// TIA Portal V20 export
// export: Created 2025-12-01T14:57:26.6752033Z, ExportSetting None, DisplayName Totally Integrated Automation Portal, DisplayVersion V20 Update 3, DisplayName TIA Portal Openness, DisplayVersion V20 Update 3, DisplayName TIA Portal Version Control Interface, DisplayVersion V20 Update 3, DisplayName STEP 7 Professional, DisplayVersion V20 Update 3, DisplayName STEP 7 Safety, DisplayVersion V20 Update 2, DisplayName WinCC Basic/Comfort/Advanced, DisplayVersion V20 Update 3, DisplayName WinCC Professional, DisplayVersion V20 Update 3, DisplayName WinCC Unified, DisplayVersion V20 Update 3
FUNCTION "FC602_ReservaPeine" : Void   // FC602, LAD
{ S7_Optimized_Access := 'TRUE' }
// stored: AutoNumber false, SetENOAutomatically false
   VAR_INPUT
      ID_Quimarox : UInt;
      ID_ElementoPeticion : UInt;
      TipoDeElemento : UInt;
   END_VAR
   VAR_OUTPUT
      NumeroPeineReservado : UInt;
   END_VAR
   VAR_TEMP
      PeineParaReserva : UInt;
      MesaFija : Bool;
      MesaMovilLateral : Bool;
      MesaMovilFrontal : Bool;
   END_VAR
BEGIN

NETWORK
TITLE = Inicializacion
/////////////////////////////////////////////////////////////////////////////////////
/////////////////////////////////////////////////////////////////////////////////////
/////////////////////////////////////////////////////////////////////////////////////
// Inicialización
      L     0;
      T     #NumeroPeineReservado;


/////////////////////////////////////////////////////////////////////////////////////
/////////////////////////////////////////////////////////////////////////////////////
/////////////////////////////////////////////////////////////////////////////////////
// Tipo de Mesa
      SET;  // Mesa Fija (1)
      L     #TipoDeElemento;
      L     1;
      ==I;
      S     #MesaFija;

      SET;  // Mesa Movil Lateral Fija (2)
      L     #TipoDeElemento;
      L     2;
      ==I;
      S     #MesaMovilLateral;


      SET;  // Mesa Movil Frontal (3)
      L     #TipoDeElemento;
      L     3;
      ==I;
      S     #MesaMovilFrontal;



NETWORK
TITLE = FASE 1 >>> Inicio de la Reserva
/////////////////////////////////////////////////////////////////////////////////////
/////////////////////////////////////////////////////////////////////////////////////
/////////////////////////////////////////////////////////////////////////////////////
// Primero miramos si hay un número de vagón valido.
// Si está a cero es que no se está ejecutando el control de posicion y no se puede reservar
      SET;
      A(;
      L     "DB602_ElementosQuimarox".Quimarox[#ID_Quimarox].Elementos[#ID_ElementoPeticion].Numero_carrier;
      L     0;  // #DatosElemento.ventana_minima
      ==I;
      );
      JC    EsperaParaReservar;


/////////////////////////////////////////////////////////////////////////////////////
/////////////////////////////////////////////////////////////////////////////////////
/////////////////////////////////////////////////////////////////////////////////////
// Miramos si el que tenemos delante >>> Aún no ha entrado en ventana , lo podríamos utilizar
      L     "DB602_ElementosQuimarox".Quimarox[#ID_Quimarox].Elementos[#ID_ElementoPeticion].Numero_carrier;
      T     #PeineParaReserva;

      SET;
      AN    "DB602_ElementosQuimarox".Quimarox[#ID_Quimarox].Elementos[#ID_ElementoPeticion].Hay_Carrier_en_ventana;
      A(;
      L     "DB602_ElementosQuimarox".Quimarox[#ID_Quimarox].Elementos[#ID_ElementoPeticion].Avance_carrier;
      L     "DB602_ElementosQuimarox".Quimarox[#ID_Quimarox].Elementos[#ID_ElementoPeticion].ventana_minima;
      <I;
      );
      JCN   FASE01_SiguientePeine;
      JU    ComprobarPeine_ParaReservar;


/////////////////////////////////////////////////////////////////////////////////////
/////////////////////////////////////////////////////////////////////////////////////
/////////////////////////////////////////////////////////////////////////////////////
/// Control de Numero de Peines
FASE01_SiguientePeine:NOP   0;
      L     "DB602_ElementosQuimarox".Quimarox[#ID_Quimarox].Elementos[#ID_ElementoPeticion].Numero_carrier;
      L     1;
      +I;
      T     #PeineParaReserva;

// comprobamos que no hemos superado el máximo de peines configurado
      SET;
      L     #PeineParaReserva;
      L     "DB600_ConfigQuimarox".Quimarox[#ID_Quimarox].datos_config.Numero_vagones;
      <=I;
      JC    ComprobarPeine_ParaReservar;

// si no hemos saltado, es que hemos superado el máximo, y tenemos que volver al peine 1
      L     1;
      T     #PeineParaReserva;
      JU    ComprobarPeine_ParaReservar;



NETWORK
TITLE = FASE 2 >>> Bucle de la Busqueda de la Reserva

/////////////////////////////////////////////////////////////////////////////////////
/////////////////////////////////////////////////////////////////////////////////////
/////////////////////////////////////////////////////////////////////////////////////
// Pasamos a comprobar el estado del carrier (vacio, habilitado, etc) para gestionar la reserva
ComprobarPeine_ParaReservar:NOP   0;



/////////////////////////////////////////////////////////////////////////////////////
/////////////////////////////////////////////////////////////////////////////////////
/////////////////////////////////////////////////////////////////////////////////////
// --- Vacio Totalmente >> NO Cargado y No Reservado
      SET;
      AN    "DB601_PeinesQuimarox".Quimarox[#ID_Quimarox].vagon[#PeineParaReserva].Carrier_Cargado;
      AN    "DB601_PeinesQuimarox".Quimarox[#ID_Quimarox].vagon[#PeineParaReserva].vagon_reservado_carga;

      AN    "DB601_PeinesQuimarox".Quimarox[#ID_Quimarox].vagon[#PeineParaReserva].vagon_cargado_SinDestino;
      AN    "DB601_PeinesQuimarox".Quimarox[#ID_Quimarox].vagon[#PeineParaReserva].carrier_no_utilizable;
      AN    "DB601_PeinesQuimarox".Quimarox[#ID_Quimarox].vagon[#PeineParaReserva].carrier_multiple;
      JC    GestionaReserva_PeineEncontrado;

// --- ESTA Cargado, pero NO Reservado >>> Para Mesa Fija
      SET;
      A     #MesaFija;
      A     "DB601_PeinesQuimarox".Quimarox[#ID_Quimarox].vagon[#PeineParaReserva].Carrier_Cargado;
      AN    "DB601_PeinesQuimarox".Quimarox[#ID_Quimarox].vagon[#PeineParaReserva].vagon_reservado_carga;

      AN    "DB601_PeinesQuimarox".Quimarox[#ID_Quimarox].vagon[#PeineParaReserva].vagon_cargado_SinDestino;
      AN    "DB601_PeinesQuimarox".Quimarox[#ID_Quimarox].vagon[#PeineParaReserva].carrier_no_utilizable;
      AN    "DB601_PeinesQuimarox".Quimarox[#ID_Quimarox].vagon[#PeineParaReserva].carrier_multiple;
      JC    GestionaReserva_PeineEncontrado;

// --- SI llega aqui, significa que el peine no se puede reservar, y tenemos que buscar en el siguiente
      JU    FASE02_BuscarSiguientePeine;


/////////////////////////////////////////////////////////////////////////////////////
/////////////////////////////////////////////////////////////////////////////////////
/////////////////////////////////////////////////////////////////////////////////////
// ese carrier no puede ser reservado y tenemos que mirar en el siguiente
FASE02_BuscarSiguientePeine:NOP   0;
      L     #PeineParaReserva;
      L     1;
      +I;
      T     #PeineParaReserva;

// comprobamos que no supera los límites
      SET;
      L     #PeineParaReserva;
      L     "DB600_ConfigQuimarox".Quimarox[#ID_Quimarox].datos_config.Numero_vagones;
      >I;
      JC    FASE02_SuperaMaximo_Peines;
      JU    FASE02_Continuar_BusquedaPeine;


/////////////////////////////////////////////////////////////////////////////////////
/////////////////////////////////////////////////////////////////////////////////////
/////////////////////////////////////////////////////////////////////////////////////
FASE02_SuperaMaximo_Peines:SET;
      L     1;
      T     #PeineParaReserva;
      JU    FASE02_Continuar_BusquedaPeine;


/////////////////////////////////////////////////////////////////////////////////////
/////////////////////////////////////////////////////////////////////////////////////
/////////////////////////////////////////////////////////////////////////////////////
// comprobamos que no hemos recorrido todos los peines intentando hacer una reserva sin exito
FASE02_Continuar_BusquedaPeine:NOP   0;
      SET;
      L     #PeineParaReserva;
      L     "DB602_ElementosQuimarox".Quimarox[#ID_Quimarox].Elementos[#ID_ElementoPeticion].Numero_carrier;
      ==I;
      JC    EsperaParaReservar;

// si no ha saltado es que tenemos que comprobar el siguiente carrier
      JU    ComprobarPeine_ParaReservar;



NETWORK
TITLE = FASE FINAL >>> Peine Encontrado >>> Activar Reserva
/////////////////////////////////////////////////////////////////////////////////////
/////////////////////////////////////////////////////////////////////////////////////
/////////////////////////////////////////////////////////////////////////////////////
// gestionamos la reserva
GestionaReserva_PeineEncontrado:NOP   0;
//      BE                         // PRUEBAS DE RESERVA CUIDADO!!!!

      SET;  // activamos el bit de reservado
      =     "DB601_PeinesQuimarox".Quimarox[#ID_Quimarox].vagon[#PeineParaReserva].vagon_reservado_carga;

// escribimos el los datos de la entrada el id del elemento que ha realizado la reserva
      L     #ID_ElementoPeticion;
      T     "DB601_PeinesQuimarox".Quimarox[#ID_Quimarox].vagon[#PeineParaReserva].punto_entrada_carga;

      L     #PeineParaReserva;
      T     #NumeroPeineReservado;

      BE;



NETWORK
TITLE = Final >>> Esperar Para Reservar
/////////////////////////////////////////////////////////////////////////////////////
// Si no hemos encontrado ningún carrier libre en el sorter, no podemos
// seguir buscando infinitamente (bucle infinito y el CPU a stop)
// tendremos que lanzar un temporizador de espera para volver a gestionar la busqueda.
EsperaParaReservar:NOP   0;
      BE;


END_FUNCTION
